PROGRAM P2_04_Cleaning_Ctrl
VAR
	bPreWash_Active					:BOOL;
	bMounting_Active				:BOOL;
	bMainClean_Active				:BOOL;
	bPWClean_Active					:BOOL;
	bRinsing_Active					:BOOL;
	bBlowing_Active					:BOOL;
	bControl_Active					:BOOL;
	
	bDischargeCloseRequest				:BOOL;
	bDischargeOpenRequest				:BOOL;
END_VAR
VAR // added by the converter: edge detectors and wires of the graphical bodies
    _w1, _w2, _w3, _w4 : BOOL;
END_VAR

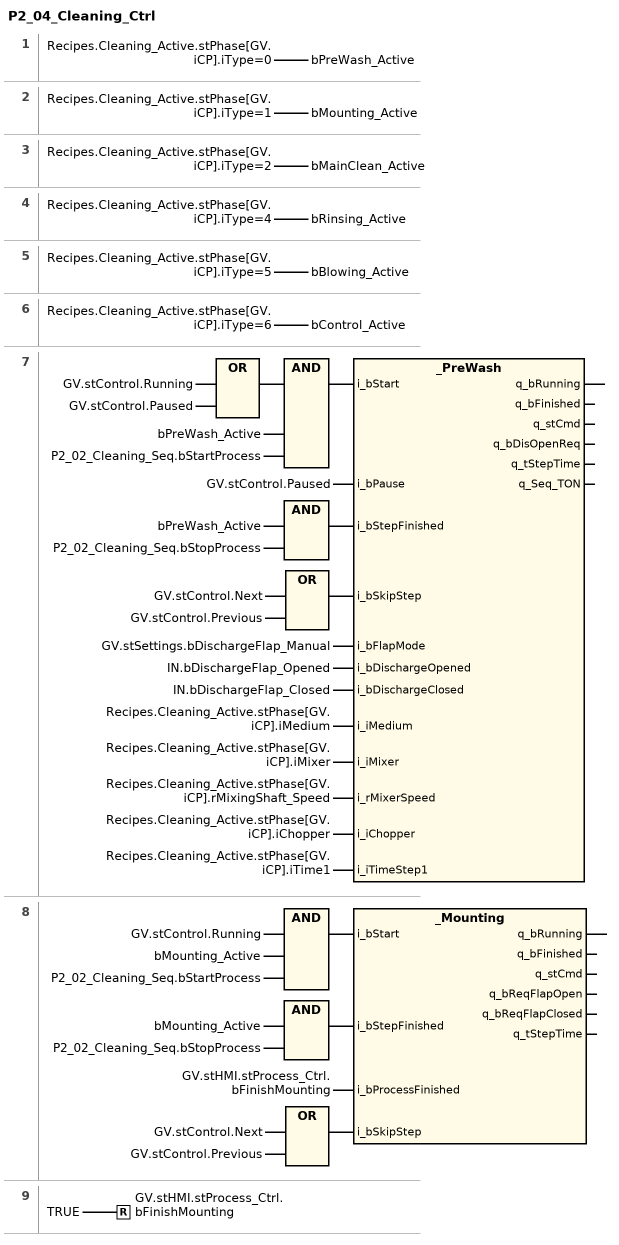
// NETWORK 1
bPreWash_Active := Recipes.Cleaning_Active.stPhase[GV.iCP].iType=0;

// NETWORK 2
bMounting_Active := Recipes.Cleaning_Active.stPhase[GV.iCP].iType=1;

// NETWORK 3
bMainClean_Active := Recipes.Cleaning_Active.stPhase[GV.iCP].iType=2;

// NETWORK 4
bRinsing_Active := Recipes.Cleaning_Active.stPhase[GV.iCP].iType=4;

// NETWORK 5
bBlowing_Active := Recipes.Cleaning_Active.stPhase[GV.iCP].iType=5;

// NETWORK 6
bControl_Active := Recipes.Cleaning_Active.stPhase[GV.iCP].iType=6;

// NETWORK 7
_PreWash(i_bStart := (GV.stControl.Running OR GV.stControl.Paused) AND bPreWash_Active AND P2_02_Cleaning_Seq.bStartProcess, i_bPause := GV.stControl.Paused, i_bStepFinished := bPreWash_Active AND P2_02_Cleaning_Seq.bStopProcess, i_bSkipStep := GV.stControl.Next OR GV.stControl.Previous, i_bFlapMode := GV.stSettings.bDischargeFlap_Manual, i_bDischargeOpened := IN.bDischargeFlap_Opened, i_bDischargeClosed := IN.bDischargeFlap_Closed, i_iMedium := Recipes.Cleaning_Active.stPhase[GV.iCP].iMedium, i_iMixer := Recipes.Cleaning_Active.stPhase[GV.iCP].iMixer, i_rMixerSpeed := Recipes.Cleaning_Active.stPhase[GV.iCP].rMixingShaft_Speed, i_iChopper := Recipes.Cleaning_Active.stPhase[GV.iCP].iChopper, i_iTimeStep1 := Recipes.Cleaning_Active.stPhase[GV.iCP].iTime1);

// NETWORK 8
_Mounting(i_bStart := GV.stControl.Running AND bMounting_Active AND P2_02_Cleaning_Seq.bStartProcess, i_bStepFinished := bMounting_Active AND P2_02_Cleaning_Seq.bStopProcess, i_bProcessFinished := GV.stHMI.stProcess_Ctrl.bFinishMounting, i_bSkipStep := GV.stControl.Next OR GV.stControl.Previous);

// NETWORK 9
GV.stHMI.stProcess_Ctrl.bFinishMounting R= TRUE;

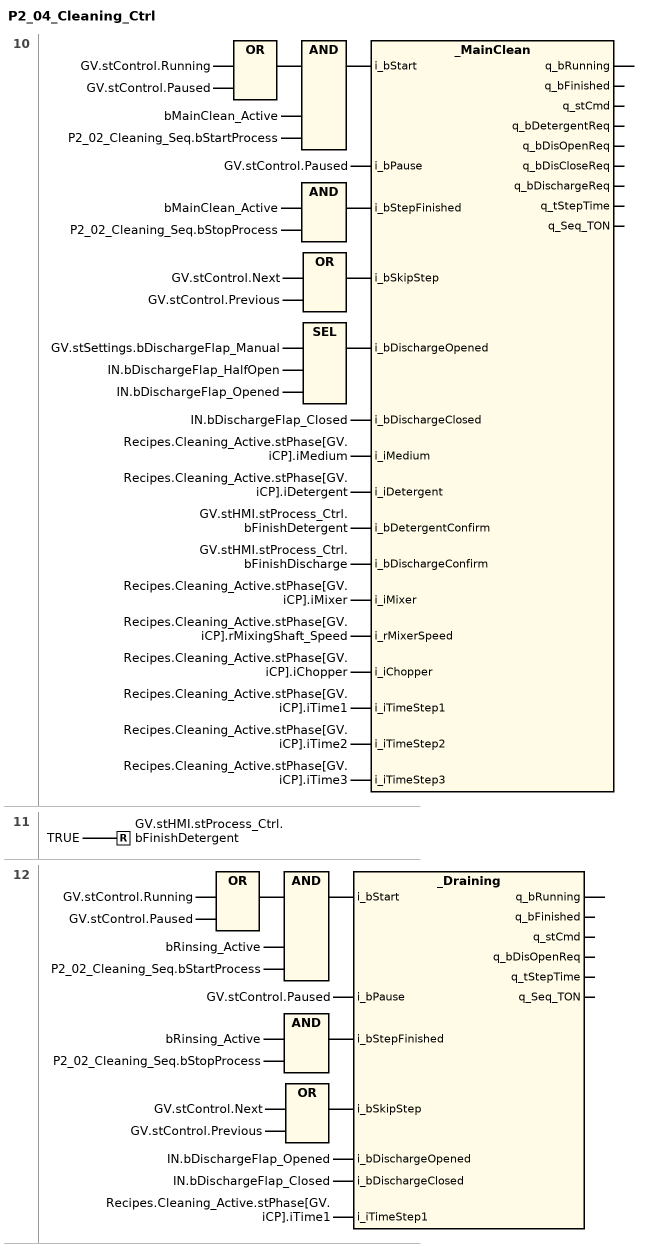
// NETWORK 10
_MainClean(i_bStart := (GV.stControl.Running OR GV.stControl.Paused) AND bMainClean_Active AND P2_02_Cleaning_Seq.bStartProcess, i_bPause := GV.stControl.Paused, i_bStepFinished := bMainClean_Active AND P2_02_Cleaning_Seq.bStopProcess, i_bSkipStep := GV.stControl.Next OR GV.stControl.Previous, i_bDischargeOpened := SEL(GV.stSettings.bDischargeFlap_Manual, IN.bDischargeFlap_HalfOpen, IN.bDischargeFlap_Opened), i_bDischargeClosed := IN.bDischargeFlap_Closed, i_iMedium := Recipes.Cleaning_Active.stPhase[GV.iCP].iMedium, i_iDetergent := Recipes.Cleaning_Active.stPhase[GV.iCP].iDetergent, i_bDetergentConfirm := GV.stHMI.stProcess_Ctrl.bFinishDetergent, i_bDischargeConfirm := GV.stHMI.stProcess_Ctrl.bFinishDischarge, i_iMixer := Recipes.Cleaning_Active.stPhase[GV.iCP].iMixer, i_rMixerSpeed := Recipes.Cleaning_Active.stPhase[GV.iCP].rMixingShaft_Speed, i_iChopper := Recipes.Cleaning_Active.stPhase[GV.iCP].iChopper, i_iTimeStep1 := Recipes.Cleaning_Active.stPhase[GV.iCP].iTime1, i_iTimeStep2 := Recipes.Cleaning_Active.stPhase[GV.iCP].iTime2, i_iTimeStep3 := Recipes.Cleaning_Active.stPhase[GV.iCP].iTime3);

// NETWORK 11
GV.stHMI.stProcess_Ctrl.bFinishDetergent R= TRUE;

// NETWORK 12
_Draining(i_bStart := (GV.stControl.Running OR GV.stControl.Paused) AND bRinsing_Active AND P2_02_Cleaning_Seq.bStartProcess, i_bPause := GV.stControl.Paused, i_bStepFinished := bRinsing_Active AND P2_02_Cleaning_Seq.bStopProcess, i_bSkipStep := GV.stControl.Next OR GV.stControl.Previous, i_bDischargeOpened := IN.bDischargeFlap_Opened, i_bDischargeClosed := IN.bDischargeFlap_Closed, i_iTimeStep1 := Recipes.Cleaning_Active.stPhase[GV.iCP].iTime1);

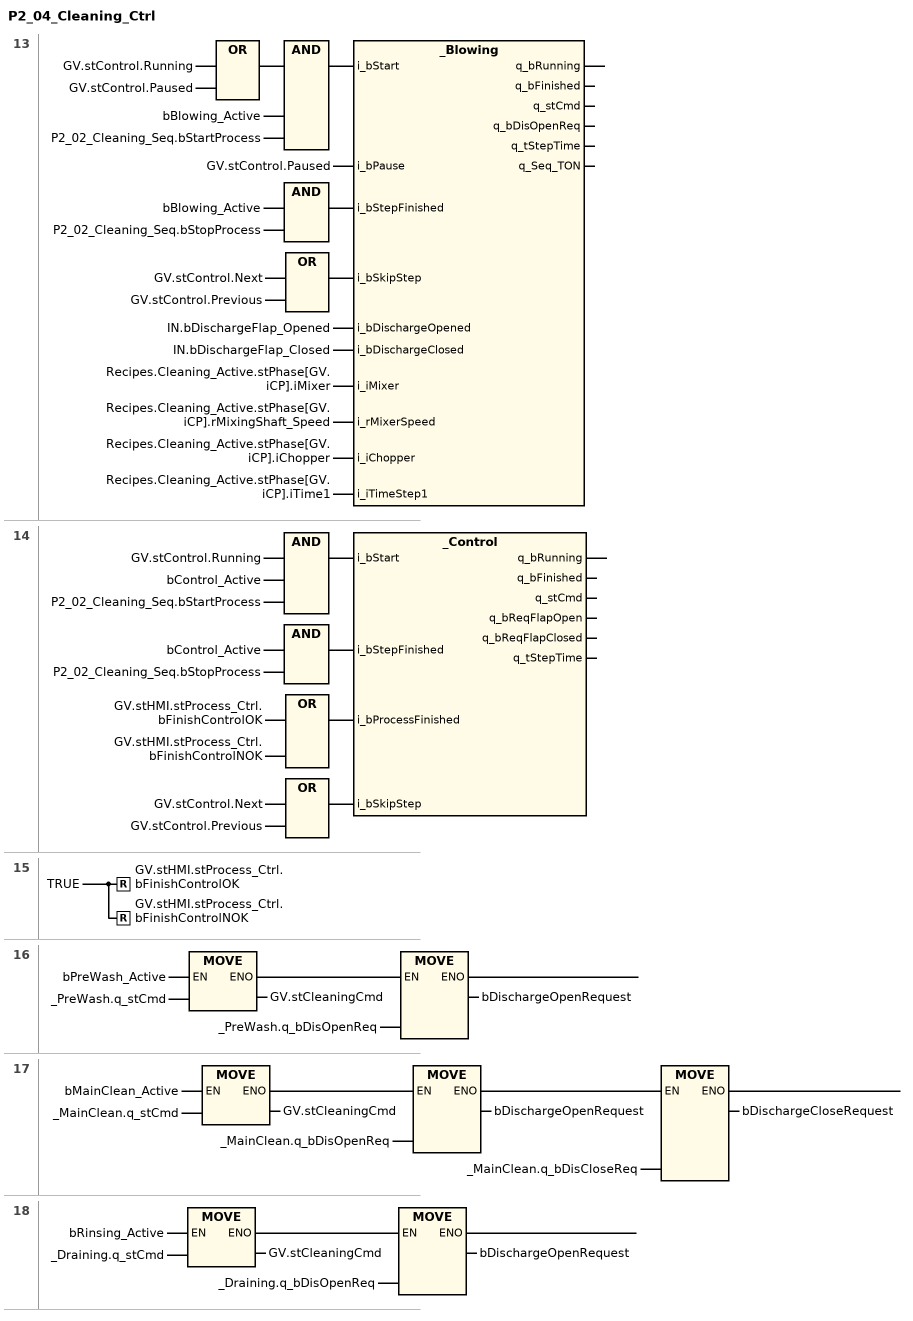
// NETWORK 13
_Blowing(i_bStart := (GV.stControl.Running OR GV.stControl.Paused) AND bBlowing_Active AND P2_02_Cleaning_Seq.bStartProcess, i_bPause := GV.stControl.Paused, i_bStepFinished := bBlowing_Active AND P2_02_Cleaning_Seq.bStopProcess, i_bSkipStep := GV.stControl.Next OR GV.stControl.Previous, i_bDischargeOpened := IN.bDischargeFlap_Opened, i_bDischargeClosed := IN.bDischargeFlap_Closed, i_iMixer := Recipes.Cleaning_Active.stPhase[GV.iCP].iMixer, i_rMixerSpeed := Recipes.Cleaning_Active.stPhase[GV.iCP].rMixingShaft_Speed, i_iChopper := Recipes.Cleaning_Active.stPhase[GV.iCP].iChopper, i_iTimeStep1 := Recipes.Cleaning_Active.stPhase[GV.iCP].iTime1);

// NETWORK 14
_Control(i_bStart := GV.stControl.Running AND bControl_Active AND P2_02_Cleaning_Seq.bStartProcess, i_bStepFinished := bControl_Active AND P2_02_Cleaning_Seq.bStopProcess, i_bProcessFinished := GV.stHMI.stProcess_Ctrl.bFinishControlOK OR GV.stHMI.stProcess_Ctrl.bFinishControlNOK, i_bSkipStep := GV.stControl.Next OR GV.stControl.Previous);

// NETWORK 15
GV.stHMI.stProcess_Ctrl.bFinishControlOK R= TRUE;
GV.stHMI.stProcess_Ctrl.bFinishControlNOK R= TRUE;

// NETWORK 16
_w1 := bPreWash_Active;
IF _w1 THEN GV.stCleaningCmd := _PreWash.q_stCmd; END_IF
IF _w1 THEN bDischargeOpenRequest := _PreWash.q_bDisOpenReq; END_IF

// NETWORK 17
_w2 := bMainClean_Active;
IF _w2 THEN GV.stCleaningCmd := _MainClean.q_stCmd; END_IF
IF _w2 THEN bDischargeOpenRequest := _MainClean.q_bDisOpenReq; END_IF
IF _w2 THEN bDischargeCloseRequest := _MainClean.q_bDisCloseReq; END_IF

// NETWORK 18
_w3 := bRinsing_Active;
IF _w3 THEN GV.stCleaningCmd := _Draining.q_stCmd; END_IF
IF _w3 THEN bDischargeOpenRequest := _Draining.q_bDisOpenReq; END_IF

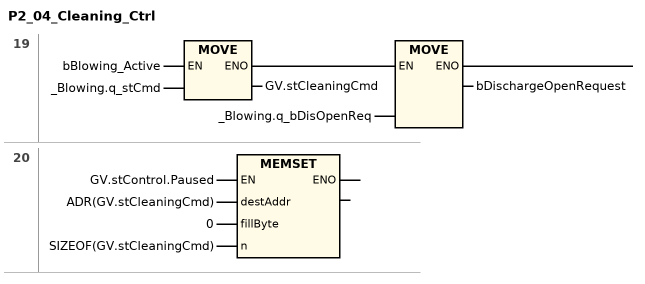
// NETWORK 19
_w4 := bBlowing_Active;
IF _w4 THEN GV.stCleaningCmd := _Blowing.q_stCmd; END_IF
IF _w4 THEN bDischargeOpenRequest := _Blowing.q_bDisOpenReq; END_IF

// NETWORK 20
IF GV.stControl.Paused THEN
    MEMSET(destAddr := ADR(GV.stCleaningCmd), fillByte := 0, n := SIZEOF(GV.stCleaningCmd));
END_IF

END_PROGRAM

(* stored: Version 1.1.0.1
   POU P2_04_Cleaning_Ctrl: Id {626edb41-8728-41d4-a27c-0fd2a6981518}, SpecialFunc None *)
